// TwinCAT 3 PLC project main
// ProgramVersion: 3.1.4024.0
// libraries:
//   Tc2_Standard, * (Beckhoff Automation GmbH)
//   Tc2_System, * (Beckhoff Automation GmbH)
//   Tc3_Module, * (Beckhoff Automation GmbH)
// project tree:
//   / GlobalTextList.TcGTLO, PlcTask.TcTTO, Visualization Manager.TcVMO (not stored)
//   POUs/ MAIN.TcPOU
//   VISUs/ Visu.TcVIS
// real-time tasks:
//   TASK PlcTask: cycle T#10ms, priority 20, ADS port 350

CONFIGURATION main
    RESOURCE PLC ON TwinCAT3
        TASK PlcTask(INTERVAL := T#10ms, PRIORITY := 20);
        PROGRAM MAIN WITH PlcTask : MAIN;
    END_RESOURCE
END_CONFIGURATION

// ---- POUs/MAIN.TcPOU
PROGRAM MAIN
VAR
	bS1 : BOOL; //Schakelaar alarm aan
	bS2 : BOOL; //Bewegins detectie
	bS3 : bool; //Reset
	
	bL1 : BOOL; //Een lamp om te tonen dat het alarm aan is
	bL2 : BOOL; //Alarm
END_VAR

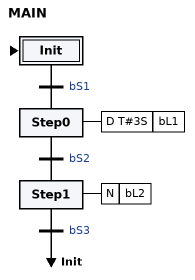
INITIAL_STEP Init:
END_STEP
TRANSITION FROM Init TO Step0
    := bS1;
END_TRANSITION
STEP Step0:
    bL1(D, T#3S);
END_STEP
TRANSITION FROM Step0 TO Step1
    := bS2;
END_TRANSITION
STEP Step1:
    bL2(N);
END_STEP
TRANSITION FROM Step1 TO Init
    := bS3;
END_TRANSITION

END_PROGRAM

// ---- GlobalTextList.TcGTLO
TEXTLIST GlobalTextList
  871 = 'Alarm'
  894 = 'Alarm gaat af'
  425 = 'Alarm staat aan'
  478 = 'bL1'
  109 = 'bL2'
  556 = 'bS1'
  150 = 'bS2'
  863 = 'bS3'
  169 = 'Label'
END_TEXTLIST

// ---- VISUs/Visu.TcVIS
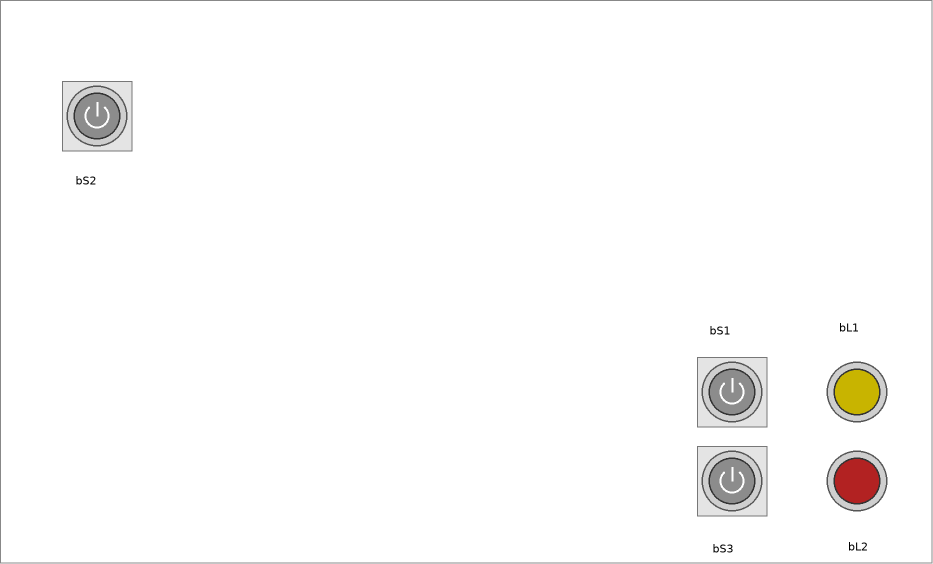
VISUALIZATION Visu  // 933x564
    Lamp1 (822,357 70x70), variable: MAIN.bL1, style: Lamp-Lamp1-Yellow
    PowerSwitch (697,357 70x70), variable: MAIN.bS1, behaviour: TAP, style: Switch-PowerSwitch-Gray
    Lamp1 (822,446 70x70), variable: MAIN.bL2, style: Lamp-Lamp1-Red
    PowerSwitch (697,446 70x70), variable: MAIN.bS3, behaviour: TAP, style: Switch-PowerSwitch-Gray
    Label (783,532 150x30), "bL2"
    Label (648,534 150x30), "bS3"
    Label (645,316 150x30), "bS1"
    Label (774,313 150x30), "bL1"
    PowerSwitch (62,81 70x70), variable: MAIN.bS2, behaviour: TAP, style: Switch-PowerSwitch-Gray
    Label (11,166 150x30), "bS2"
END_VISUALIZATION
